# B&R Automation Studio project SDCAxis (part 2)

#### gmcipiec.cnc
```
Root (LangModule=ailgcode, Version=1.0)
  AxesSpec
  PrimTypes (PatternSuffix=:[^\d\w$#])
    BOOL (BRType=BOOL)
    STRING (BRType=STRING)
    WSTRING (BRType=WSTRING)
    TIME (BRType=TIME)
    SINT (BRType=SINT)
    INT (BRType=INT)
    DINT (BRType=DINT)
    USINT (BRType=USINT)
    UINT (BRType=UINT)
    UDINT (BRType=UDINT)
    REAL (BRType=REAL)
    LREAL (BRType=LREAL)
    DATE (BRType=DATE)
    DATE_AND_TIME (BRType=DATE_AND_TIME)
    DT (BRType=DT)
    TIME_OF_DAY (BRType=TIME_OF_DAY)
    TOD (BRType=TIME_OF_DAY)
    BYTE (BRType=BYTE)
    WORD (BRType=WORD)
    DWORD (BRType=DWORD)
  BuiltInProcs:
    SetCyclicId = #job->group_id = $[1]; (MinArgs=1, MaxArgs=1, Eval=Early)
    WaitForCyclic = if ( Defined(:$[1]:) ) 
        WaitForCyclicGroups(:${*}:);  
      else
        WaitForCyclicJob(:#last_job_id:);
      endif (MinArgs=0, MaxArgs=*)
    REPORT (MinArgs=2, MaxArgs=2)
      Arg (ref=id, DataType=INT)
      Arg (ref=msg, DataType=STRING)
    WARN (MinArgs=2, MaxArgs=2)
      Arg (ref=id, DataType=INT)
      Arg (ref=msg, DataType=STRING)
    HALT (MinArgs=2, MaxArgs=2)
      Arg (ref=id, DataType=INT)
      Arg (ref=msg, DataType=STRING)
    ERROR (MinArgs=2, MaxArgs=2)
      Arg (ref=id, DataType=INT)
      Arg (ref=msg, DataType=STRING)
    LOADBG (MinArgs=1, MaxArgs=1)
      Arg (ref=filename, DataType=STRING)
    LOAD (MinArgs=1, MaxArgs=1)
      Arg (ref=filename, DataType=STRING)
    UNLOAD (MinArgs=1, MaxArgs=1)
      Arg (ref=filename, DataType=STRING)
    EXEC (MinArgs=1, MaxArgs=5)
      Arg (ref=filename, DataType=STRING)
      Arg (ref=arguments, DataType=ANY_DATA)
      Arg (ref=langId, DataType=INT)
      Arg (ref=block, DataType=INT, MinCount=0, MaxCount=1, DenyArgs=5, WriteOpts=:)
      Arg (ref=line, DataType=INT, MinCount=0, MaxCount=1, DenyArgs=4, WriteOpts=:)
    EXEC_RPC (MinArgs=2, MaxArgs=4)
      Arg (ref=filename, DataType=STRING)
      Arg (ref=arguments, DataType=ANY_DATA)
      Arg (ref=langId, DataType=INT)
      Arg (ref=rpc, DataType=ANY_DATA, MinCount=1, MaxCount=1)
    EVAL (MinArgs=1, MaxArgs=2)
      Arg (ref=expression, DataType=STRING)
      Arg (ref=langId, DataType=INT)
    PUSH_PACKET = PushPacket(::);
    PUSH_PACKET_CMD (MinArgs=1, MaxArgs=2)
      Arg (ref=cmd, DataType=INT)
      Arg (ref=data, DataType=ANY_DATA)
    DISPATCH_AND_WAIT (MinArgs=1, MaxArgs=1)
      Arg (ref=cmd, DataType=INT)
    START_PACKET_LIST = #inhibit_mp_list_dispatch = 1;
    END_PACKET_LIST = #inhibit_mp_list_dispatch = 0;
    LOG_INFO (MinArgs=1, MaxArgs=1)
      Arg (ref=msg, DataType=STRING)
    SET_BLOCK_NUMBER = SetCurBlockNr(:$[1]:); (MinArgs=1, MaxArgs=1)
    SBLOF_PATH = #next_motion.Command = MPCMD_SBL_PATH_INHIBIT;
      PushPacket(::);
    SBLON_PATH = #next_motion.Command = MPCMD_SBL_PATH_RELEASE;
      PushPacket(::);
  BuiltInFns:
    ABS = Abs(:$[1]:) (ReturnType=ANY_NUM, ArgType1=ANY_NUM, Inline=Yes)
    SIN = RSin(:$[1]:) (ReturnType=ANY_REAL, ArgType1=ANY_REAL, Inline=Yes)
    COS = RCos(:$[1]:) (ReturnType=ANY_REAL, ArgType1=ANY_REAL, Inline=Yes)
    TAN = RTan(:$[1]:) (ReturnType=ANY_REAL, ArgType1=ANY_REAL, Inline=Yes)
    ASIN = RASin(:$[1]:) (ReturnType=ANY_REAL, ArgType1=ANY_REAL, Inline=Yes)
    ACOS = RACos(:$[1]:) (ReturnType=ANY_REAL, ArgType1=ANY_REAL, Inline=Yes)
    ATAN = RATan(:$[1]:) (ReturnType=ANY_REAL, ArgType1=ANY_REAL, Inline=Yes)
    SQRT = Sqrt(:$[1]:) (ReturnType=ANY_REAL, ArgType1=ANY_REAL, Inline=Yes)
    LN = Ln(:$[1]:) (ReturnType=ANY_REAL, ArgType1=ANY_REAL, Inline=Yes)
    EXP = Exp(:$[1]:) (ReturnType=ANY_REAL, ArgType1=ANY_REAL, Inline=Yes)
    LOG = Log(:$[1]:) (ReturnType=ANY_REAL, ArgType1=ANY_REAL, Inline=Yes)
    EXPT = Pow(:$[1],$[2]:) (ReturnType=ANY_REAL, ArgType1=ANY_REAL, ArgType2=ANY_NUM, Inline=Yes)
    TRUNC = ToInt(:Fix(:$[1]:):) (ReturnType=IEC_INT, ArgType1=ANY_REAL, Inline=Yes)
    ADR = Adr(:\$[1]:) (ReturnType=IEC_UDINT, ArgType1=ANY_DATA, Inline=Yes)
    REF = \$[1] (ReturnType=ANY_DATA, ArgType1=ANY_DATA, Inline=Yes)
    SIZEOF = Sizeof(:\$[1]:) (ReturnType=IEC_UINT, NumArgs=1, Inline=Yes)
    LIMIT (ReturnType=ANY_NUM, Inline=No)
      Arg (ref=MIN, DataType=ANY_NUM)
      Arg (ref=IN, DataType=ANY_NUM)
      Arg (ref=MAX, DataType=ANY_NUM)
    MIN (ReturnType=ANY_NUM, Inline=No)
      Arg (ref=IN1, DataType=ANY_NUM)
      Arg (ref=IN2, DataType=ANY_NUM)
    MAX (ReturnType=ANY_NUM, Inline=No)
      Arg (ref=IN1, DataType=ANY_NUM)
      Arg (ref=IN2, DataType=ANY_NUM)
    ROL = BitRotL(:$[1],$[2]:) (ReturnType=ANY_NUM, ArgType1=ANY_NUM, ArgType2=IEC_SINT)
    ROR = BitRotR(:$[1],$[2]:) (ReturnType=ANY_NUM, ArgType1=ANY_NUM, ArgType2=IEC_SINT)
    SHR = BitShR(:$[1],$[2]:) (ReturnType=ANY_NUM, ArgType1=ANY_NUM, ArgType2=IEC_SINT)
    SHL = BitShL(:$[1],$[2]:) (ReturnType=ANY_NUM, ArgType1=ANY_NUM, ArgType2=IEC_SINT)
    BIT_TST = AsBitTst(:$[1],$[2]:) (ReturnType=ANY_NUM, ArgType1=ANY_NUM, ArgType2=IEC_SINT)
    BIT_SET = AsBitSet(:$[1],$[2]:) (ReturnType=ANY_NUM, ArgType1=ANY_NUM, ArgType2=IEC_SINT)
    BIT_CLR = AsBitClr(:$[1],$[2]:) (ReturnType=ANY_NUM, ArgType1=ANY_NUM, ArgType2=IEC_SINT)
    TO_BOOL = ToBool(:$[1]:) (ReturnType=IEC_BOOL, ArgType1=ANY_DATA, Inline=Yes)
    TO_USINT = ToUInt(:$[1],1:) (ReturnType=IEC_USINT, ArgType1=ANY_DATA, Inline=Yes)
    TO_BYTE = ToUInt(:$[1],1:) (ReturnType=IEC_BYTE, ArgType1=ANY_DATA, Inline=Yes)
    TO_SINT = ToInt(:$[1],1:) (ReturnType=IEC_SINT, ArgType1=ANY_DATA, Inline=Yes)
    TO_UINT = ToUInt(:$[1],2:) (ReturnType=IEC_UINT, ArgType1=ANY_DATA, Inline=Yes)
    TO_WORD = ToUInt(:$[1],2:) (ReturnType=IEC_WORD, ArgType1=ANY_DATA, Inline=Yes)
    TO_INT = ToInt(:$[1],2:) (ReturnType=IEC_INT, ArgType1=ANY_DATA, Inline=Yes)
    TO_UDINT = ToUInt(:$[1]:) (ReturnType=IEC_UDINT, ArgType1=ANY_DATA, Inline=Yes)
    TO_DWORD = ToUInt(:$[1]:) (ReturnType=IEC_DWORD, ArgType1=ANY_DATA, Inline=Yes)
    TO_DINT = ToInt(:$[1]:) (ReturnType=IEC_DINT, ArgType1=ANY_DATA, Inline=Yes)
    TO_TIME = ToTime(:$[1]:) (ReturnType=IEC_TIME, ArgType1=ANY_DATA, Inline=Yes)
    TO_DT = ToDT(:$[1]:) (ReturnType=IEC_DT, ArgType1=ANY_DATA, Inline=Yes)
    TO_DATE_AND_TIME = ToDT(:$[1]:) (ReturnType=IEC_DT, ArgType1=ANY_DATA, Inline=Yes)
    TO_TOD = ToTOD(:$[1]:) (ReturnType=IEC_TOD, ArgType1=ANY_DATA, Inline=Yes)
    TO_TIME_OF_DAY = ToTOD(:$[1]:) (ReturnType=IEC_TOD, ArgType1=ANY_DATA, Inline=Yes)
    TO_DATE = ToDate(:$[1]:) (ReturnType=IEC_DATE, ArgType1=ANY_DATA, Inline=Yes)
    TO_REAL = ToFloat(:$[1]:) (ReturnType=IEC_REAL, ArgType1=ANY_DATA, Inline=Yes)
    TO_LREAL = ToLReal(:$[1]:) (ReturnType=IEC_LREAL, ArgType1=ANY_DATA, Inline=Yes)
    TO_STRING = ToString(:$[1]:) (ReturnType=IEC_STRING, ArgType1=ANY_DATA, Inline=Yes)
    TO_WSTRING = ToWString(:$[1]:) (ReturnType=IEC_WSTRING, ArgType1=ANY_DATA, Inline=Yes)
    USINT_TO_BOOL = ToBool(:$[1]:) (ReturnType=IEC_BOOL, ArgType1=IEC_USINT, Inline=Yes)
    SINT_TO_BOOL = ToBool(:$[1]:) (ReturnType=IEC_BOOL, ArgType1=IEC_SINT, Inline=Yes)
    UINT_TO_BOOL = ToBool(:$[1]:) (ReturnType=IEC_BOOL, ArgType1=IEC_UINT, Inline=Yes)
    INT_TO_BOOL = ToBool(:$[1]:) (ReturnType=IEC_BOOL, ArgType1=IEC_INT, Inline=Yes)
    UDINT_TO_BOOL = ToBool(:$[1]:) (ReturnType=IEC_BOOL, ArgType1=IEC_UDINT, Inline=Yes)
    DINT_TO_BOOL = ToBool(:$[1]:) (ReturnType=IEC_BOOL, ArgType1=IEC_DINT, Inline=Yes)
    REAL_TO_BOOL = ToBool(:$[1]:) (ReturnType=IEC_BOOL, ArgType1=IEC_REAL, Inline=Yes)
    LREAL_TO_BOOL = ToBool(:$[1]:) (ReturnType=IEC_BOOL, ArgType1=IEC_LREAL, Inline=Yes)
    TIME_TO_BOOL = ToBool(:$[1]:) (ReturnType=IEC_BOOL, ArgType1=IEC_TIME, Inline=Yes)
    DT_TO_BOOL = ToBool(:$[1]:) (ReturnType=IEC_BOOL, ArgType1=IEC_DT, Inline=Yes)
    TOD_TO_BOOL = ToBool(:$[1]:) (ReturnType=IEC_BOOL, ArgType1=IEC_TOD, Inline=Yes)
    BYTE_TO_BOOL = ToBool(:$[1]:) (ReturnType=IEC_BOOL, ArgType1=IEC_BYTE, Inline=Yes)
    WORD_TO_BOOL = ToBool(:$[1]:) (ReturnType=IEC_BOOL, ArgType1=IEC_WORD, Inline=Yes)
    DWORD_TO_BOOL = ToBool(:$[1]:) (ReturnType=IEC_BOOL, ArgType1=IEC_DWORD, Inline=Yes)
    BOOL_TO_USINT = ToUInt(:$[1],1:) (ReturnType=IEC_USINT, ArgType1=IEC_BOOL, Inline=Yes)
    SINT_TO_USINT = ToUInt(:$[1],1:) (ReturnType=IEC_USINT, ArgType1=IEC_SINT, Inline=Yes)
    UINT_TO_USINT = ToUInt(:$[1],1:) (ReturnType=IEC_USINT, ArgType1=IEC_UINT, Inline=Yes)
    INT_TO_USINT = ToUInt(:$[1],1:) (ReturnType=IEC_USINT, ArgType1=IEC_INT, Inline=Yes)
    UDINT_TO_USINT = ToUInt(:$[1],1:) (ReturnType=IEC_USINT, ArgType1=IEC_UDINT, Inline=Yes)
    DINT_TO_USINT = ToUInt(:$[1],1:) (ReturnType=IEC_USINT, ArgType1=IEC_DINT, Inline=Yes)
    REAL_TO_USINT = ToUInt(:$[1],1:) (ReturnType=IEC_USINT, ArgType1=IEC_REAL, Inline=Yes)
    LREAL_TO_USINT = ToUInt(:$[1],1:) (ReturnType=IEC_USINT, ArgType1=IEC_LREAL, Inline=Yes)
    BOOL_TO_SINT = ToInt(:$[1],1:) (ReturnType=IEC_SINT, ArgType1=IEC_BOOL, Inline=Yes)
    USINT_TO_SINT = ToInt(:$[1],1:) (ReturnType=IEC_SINT, ArgType1=IEC_USINT, Inline=Yes)
    UINT_TO_SINT = ToInt(:$[1],1:) (ReturnType=IEC_SINT, ArgType1=IEC_UINT, Inline=Yes)
    INT_TO_SINT = ToInt(:$[1],1:) (ReturnType=IEC_SINT, ArgType1=IEC_INT, Inline=Yes)
    UDINT_TO_SINT = ToInt(:$[1],1:) (ReturnType=IEC_SINT, ArgType1=IEC_UDINT, Inline=Yes)
    DINT_TO_SINT = ToInt(:$[1],1:) (ReturnType=IEC_SINT, ArgType1=IEC_DINT, Inline=Yes)
    REAL_TO_SINT = ToInt(:$[1],1:) (ReturnType=IEC_SINT, ArgType1=IEC_REAL, Inline=Yes)
    LREAL_TO_SINT = ToInt(:$[1],1:) (ReturnType=IEC_SINT, ArgType1=IEC_LREAL, Inline=Yes)
    BOOL_TO_UINT = ToUInt(:$[1],2:) (ReturnType=IEC_UINT, ArgType1=IEC_BOOL, Inline=Yes)
    SINT_TO_UINT = ToUInt(:$[1],2:) (ReturnType=IEC_UINT, ArgType1=IEC_SINT, Inline=Yes)
    USINT_TO_UINT = ToUInt(:$[1],2:) (ReturnType=IEC_UINT, ArgType1=IEC_USINT, Inline=Yes)
    INT_TO_UINT = ToUInt(:$[1],2:) (ReturnType=IEC_UINT, ArgType1=IEC_INT, Inline=Yes)
    UDINT_TO_UINT = ToUInt(:$[1],2:) (ReturnType=IEC_UINT, ArgType1=IEC_UDINT, Inline=Yes)
    DINT_TO_UINT = ToUInt(:$[1],2:) (ReturnType=IEC_UINT, ArgType1=IEC_DINT, Inline=Yes)
    REAL_TO_UINT = ToUInt(:$[1],2:) (ReturnType=IEC_UINT, ArgType1=IEC_REAL, Inline=Yes)
    LREAL_TO_UINT = ToUInt(:$[1],2:) (ReturnType=IEC_UINT, ArgType1=IEC_LREAL, Inline=Yes)
    BOOL_TO_INT = ToInt(:$[1],2:) (ReturnType=IEC_INT, ArgType1=IEC_BOOL, Inline=Yes)
    SINT_TO_INT = ToInt(:$[1],2:) (ReturnType=IEC_INT, ArgType1=IEC_SINT, Inline=Yes)
    USINT_TO_INT = ToInt(:$[1],2:) (ReturnType=IEC_INT, ArgType1=IEC_USINT, Inline=Yes)
    UINT_TO_INT = ToInt(:$[1],2:) (ReturnType=IEC_INT, ArgType1=IEC_UINT, Inline=Yes)
    UDINT_TO_INT = ToInt(:$[1],2:) (ReturnType=IEC_INT, ArgType1=IEC_UDINT, Inline=Yes)
    DINT_TO_INT = ToInt(:$[1],2:) (ReturnType=IEC_INT, ArgType1=IEC_DINT, Inline=Yes)
    REAL_TO_INT = ToInt(:$[1],2:) (ReturnType=IEC_INT, ArgType1=IEC_REAL, Inline=Yes)
    LREAL_TO_INT = ToInt(:$[1],2:) (ReturnType=IEC_INT, ArgType1=IEC_LREAL, Inline=Yes)
    BOOL_TO_UDINT = ToUInt(:$[1]:) (ReturnType=IEC_UDINT, ArgType1=IEC_BOOL, Inline=Yes)
    USINT_TO_UDINT = ToUInt(:$[1]:) (ReturnType=IEC_UDINT, ArgType1=IEC_USINT, Inline=Yes)
    SINT_TO_UDINT = ToUInt(:$[1]:) (ReturnType=IEC_UDINT, ArgType1=IEC_SINT, Inline=Yes)
    UINT_TO_UDINT = ToUInt(:$[1]:) (ReturnType=IEC_UDINT, ArgType1=IEC_UINT, Inline=Yes)
    INT_TO_UDINT = ToUInt(:$[1]:) (ReturnType=IEC_UDINT, ArgType1=IEC_INT, Inline=Yes)
    DINT_TO_UDINT = ToUInt(:$[1]:) (ReturnType=IEC_UDINT, ArgType1=IEC_DINT, Inline=Yes)
    REAL_TO_UDINT = ToUInt(:$[1]:) (ReturnType=IEC_UDINT, ArgType1=IEC_REAL, Inline=Yes)
    LREAL_TO_UDINT = ToUInt(:$[1]:) (ReturnType=IEC_UDINT, ArgType1=IEC_LREAL, Inline=Yes)
    TIME_TO_UDINT = ToUInt(:$[1]:) (ReturnType=IEC_UDINT, ArgType1=IEC_TIME, Inline=Yes)
    DT_TO_UDINT = ToUInt(:$[1]:) (ReturnType=IEC_UDINT, ArgType1=IEC_DT, Inline=Yes)
    BOOL_TO_DINT = ToInt(:$[1]:) (ReturnType=IEC_DINT, ArgType1=IEC_BOOL, Inline=Yes)
    USINT_TO_DINT = ToInt(:$[1]:) (ReturnType=IEC_DINT, ArgType1=IEC_USINT, Inline=Yes)
    SINT_TO_DINT = ToInt(:$[1]:) (ReturnType=IEC_DINT, ArgType1=IEC_SINT, Inline=Yes)
    UINT_TO_DINT = ToInt(:$[1]:) (ReturnType=IEC_DINT, ArgType1=IEC_UINT, Inline=Yes)
    INT_TO_DINT = ToInt(:$[1]:) (ReturnType=IEC_DINT, ArgType1=IEC_INT, Inline=Yes)
    UDINT_TO_DINT = ToInt(:$[1]:) (ReturnType=IEC_DINT, ArgType1=IEC_UDINT, Inline=Yes)
    REAL_TO_DINT = ToInt(:$[1]:) (ReturnType=IEC_DINT, ArgType1=IEC_REAL, Inline=Yes)
    LREAL_TO_DINT = ToInt(:$[1]:) (ReturnType=IEC_DINT, ArgType1=IEC_LREAL, Inline=Yes)
    TIME_TO_DINT = ToInt(:$[1]:) (ReturnType=IEC_DINT, ArgType1=IEC_TIME, Inline=Yes)
    DT_TO_DINT = ToInt(:$[1]:) (ReturnType=IEC_DINT, ArgType1=IEC_DT, Inline=Yes)
    BOOL_TO_TIME = ToTime(:$[1]:) (ReturnType=IEC_TIME, ArgType1=IEC_BOOL, Inline=Yes)
    DINT_TO_TIME = ToTime(:$[1]:) (ReturnType=IEC_TIME, ArgType1=IEC_DINT, Inline=Yes)
    UDINT_TO_TIME = ToTime(:$[1]:) (ReturnType=IEC_TIME, ArgType1=IEC_UDINT, Inline=Yes)
    BOOL_TO_DT = ToDT(:$[1]:) (ReturnType=IEC_DT, ArgType1=IEC_BOOL, Inline=Yes)
    DINT_TO_DT = ToDT(:$[1]:) (ReturnType=IEC_DT, ArgType1=IEC_DINT, Inline=Yes)
    UDINT_TO_DT = ToDT(:$[1]:) (ReturnType=IEC_DT, ArgType1=IEC_UDINT, Inline=Yes)
    BOOL_TO_REAL = ToFloat(:$[1]:) (ReturnType=IEC_REAL, ArgType1=IEC_BOOL, Inline=Yes)
    USINT_TO_REAL = ToFloat(:$[1]:) (ReturnType=IEC_REAL, ArgType1=IEC_USINT, Inline=Yes)
    SINT_TO_REAL = ToFloat(:$[1]:) (ReturnType=IEC_REAL, ArgType1=IEC_SINT, Inline=Yes)
    UINT_TO_REAL = ToFloat(:$[1]:) (ReturnType=IEC_REAL, ArgType1=IEC_UINT, Inline=Yes)
    INT_TO_REAL = ToFloat(:$[1]:) (ReturnType=IEC_REAL, ArgType1=IEC_INT, Inline=Yes)
    UDINT_TO_REAL = ToFloat(:$[1]:) (ReturnType=IEC_REAL, ArgType1=IEC_UDINT, Inline=Yes)
    DINT_TO_REAL = ToFloat(:$[1]:) (ReturnType=IEC_REAL, ArgType1=IEC_DINT, Inline=Yes)
    LREAL_TO_REAL = ToFloat(:$[1]:) (ReturnType=IEC_REAL, ArgType1=IEC_LREAL, Inline=Yes)
    TIME_TO_REAL = ToFloat(:$[1]:) (ReturnType=IEC_REAL, ArgType1=IEC_TIME, Inline=Yes)
    BOOL_TO_LREAL = ToLReal(:$[1]:) (ReturnType=IEC_LREAL, ArgType1=IEC_BOOL, Inline=Yes)
    USINT_TO_LREAL = ToLReal(:$[1]:) (ReturnType=IEC_LREAL, ArgType1=IEC_USINT, Inline=Yes)
    SINT_TO_LREAL = ToLReal(:$[1]:) (ReturnType=IEC_LREAL, ArgType1=IEC_SINT, Inline=Yes)
    UINT_TO_LREAL = ToLReal(:$[1]:) (ReturnType=IEC_LREAL, ArgType1=IEC_UINT, Inline=Yes)
    INT_TO_LREAL = ToLReal(:$[1]:) (ReturnType=IEC_LREAL, ArgType1=IEC_INT, Inline=Yes)
    UDINT_TO_LREAL = ToLReal(:$[1]:) (ReturnType=IEC_LREAL, ArgType1=IEC_UDINT, Inline=Yes)
    DINT_TO_LREAL = ToLReal(:$[1]:) (ReturnType=IEC_LREAL, ArgType1=IEC_DINT, Inline=Yes)
    REAL_TO_LREAL = ToLReal(:$[1]:) (ReturnType=IEC_LREAL, ArgType1=IEC_REAL, Inline=Yes)
    TIME_TO_LREAL = ToLReal(:$[1]:) (ReturnType=IEC_LREAL, ArgType1=IEC_TIME, Inline=Yes)
    BOOL_TO_STRING = ToString(:ToBool(:$[1]:):) (ReturnType=IEC_STRING, ArgType1=IEC_BOOL, Inline=Yes)
    USINT_TO_STRING = ToString(:ToUInt(:$[1],1:):) (ReturnType=IEC_STRING, ArgType1=IEC_USINT, Inline=Yes)
    SINT_TO_STRING = ToString(:ToInt(:$[1],1:):) (ReturnType=IEC_STRING, ArgType1=IEC_SINT, Inline=Yes)
    UINT_TO_STRING = ToString(:ToUInt(:$[1],2:):) (ReturnType=IEC_STRING, ArgType1=IEC_UINT, Inline=Yes)
    INT_TO_STRING = ToString(:ToInt(:$[1],2:):) (ReturnType=IEC_STRING, ArgType1=IEC_INT, Inline=Yes)
    UDINT_TO_STRING = ToString(:ToUInt(:$[1]:):) (ReturnType=IEC_STRING, ArgType1=IEC_UDINT, Inline=Yes)
    DINT_TO_STRING = ToString(:ToInt(:$[1]:):) (ReturnType=IEC_STRING, ArgType1=IEC_DINT, Inline=Yes)
    REAL_TO_STRING = ToString(:ToFloat(:$[1]:):) (ReturnType=IEC_STRING, ArgType1=IEC_REAL, Inline=Yes)
    LREAL_TO_STRING = ToString(:ToLReal(:$[1]:):) (ReturnType=IEC_STRING, ArgType1=IEC_LREAL, Inline=Yes)
    STRING_TO_BOOL = ToBool(:StrToInt(:$[1]:):) (ReturnType=IEC_BOOL, ArgType1=IEC_STRING, Inline=Yes)
    STRING_TO_USINT = ToUInt(:StrToInt(:$[1]:),1:) (ReturnType=IEC_USINT, ArgType1=IEC_STRING, Inline=Yes)
    STRING_TO_SINT = ToInt(:StrToInt(:$[1]:),1:) (ReturnType=IEC_SINT, ArgType1=IEC_STRING, Inline=Yes)
    STRING_TO_UINT = ToUInt(:StrToInt(:$[1]:),2:) (ReturnType=IEC_UINT, ArgType1=IEC_STRING, Inline=Yes)
    STRING_TO_INT = ToInt(:StrToInt(:$[1]:),2:) (ReturnType=IEC_INT, ArgType1=IEC_STRING, Inline=Yes)
    STRING_TO_UDINT = ToUInt(:StrToInt(:$[1]:):) (ReturnType=IEC_UDINT, ArgType1=IEC_STRING, Inline=Yes)
    STRING_TO_DINT = ToInt(:StrToInt(:$[1]:):) (ReturnType=IEC_DINT, ArgType1=IEC_STRING, Inline=Yes)
    STRING_TO_REAL = ToFloat(:ToLReal(:$[1]:):) (ReturnType=IEC_REAL, ArgType1=IEC_STRING, Inline=Yes)
    STRING_TO_LREAL = ToLReal(:$[1]:) (ReturnType=IEC_LREAL, ArgType1=IEC_STRING, Inline=Yes)
    LEN = __LEN(:$[1]:) (ReturnType=IEC_INT, ArgType1=IEC_STRING, Inline=Yes)
    LEFT = __LEFT(:$[1], $[2]:) (ReturnType=IEC_STRING, ArgType1=IEC_STRING, ArgType2=IEC_INT, Inline=Yes)
    RIGHT = __RIGHT(:$[1], $[2]:) (ReturnType=IEC_STRING, ArgType1=IEC_STRING, ArgType2=IEC_INT, Inline=Yes)
    MID = __MID(:$[1], $[2], $[3]:) (ReturnType=IEC_STRING, ArgType1=IEC_STRING, ArgType2=IEC_INT, ArgType3=IEC_INT, Inline=Yes)
    CONCAT = __CONCAT(:$[1], $[2]:) (ReturnType=IEC_STRING, ArgType1=IEC_STRING, ArgType2=IEC_STRING, Inline=Yes)
    INSERT = __INSERT(:$[1], $[2], $[3]:) (ReturnType=IEC_STRING, ArgType1=IEC_STRING, ArgType2=IEC_STRING, ArgType3=IEC_INT, Inline=Yes)
    DELETE = __DELETE(:$[1], $[2], $[3]:) (ReturnType=IEC_STRING, ArgType1=IEC_STRING, ArgType2=IEC_INT, ArgType3=IEC_INT, Inline=Yes)
    REPLACE = __REPLACE(:$[1], $[2], $[3], $[4]:) (ReturnType=IEC_STRING, ArgType1=IEC_STRING, ArgType2=IEC_STRING, ArgType3=IEC_INT, ArgType4=IEC_INT, Inline=Yes)
    FIND = __FIND(:$[1], $[2]:) (ReturnType=IEC_INT, ArgType1=IEC_STRING, ArgType2=IEC_STRING, Inline=Yes)
    IP_INST_NUM = IpInstNum(::) (ReturnType=IEC_INT, NumArgs=0)
    IP_OWNER_ID = IpOwnerId(::) (ReturnType=IEC_INT, NumArgs=0)
    PACKET_DATA_ADR = GetIpInt(:6:) (ReturnType=IEC_UDINT, NumArgs=0, Inline=Yes)
    PACKET_COMMAND_ADR = GetIpInt(:7:) (ReturnType=IEC_UDINT, NumArgs=0, Inline=Yes)
  Parameters:
    QUOTED (QuotedName=$R, ValueType=FLOAT, ReturnType=IEC_LREAL)
      ARG (ref=EXPR, DataType=INT, MinValue=0, MaxValue=999)
    QUOTED (QuotedName=$P, ValueType=FLOAT, ReturnType=IEC_LREAL)
      ARG (ref=EXPR, DataType=INT, MinValue=0, MaxValue=999)
    QUOTED (QuotedName=$EXB, ValueType=INT, ReturnType=IEC_SINT)
      ARG (ref=EXPR, DataType=INT, MinValue=0, MaxValue=99)
    QUOTED (QuotedName=$EXW, ValueType=INT, ReturnType=IEC_INT)
      ARG (ref=EXPR, DataType=INT, MinValue=0, MaxValue=99)
    QUOTED (QuotedName=$EXL, ValueType=INT, ReturnType=IEC_DINT)
      ARG (ref=EXPR, DataType=INT, MinValue=0, MaxValue=99)
    QUOTED (QuotedName=$EXF, ValueType=FLOAT, ReturnType=IEC_REAL)
      ARG (ref=EXPR, DataType=INT, MinValue=0, MaxValue=3999)
    QUOTED (QuotedName=$MW, Synchronous=Yes, ValueType=INT, ReturnType=IEC_INT)
      ARG (ref=EXPR, DataType=INT, MinValue=0, MaxValue=99)
    QUOTED (QuotedName=$ML, Synchronous=Yes, ValueType=INT, ReturnType=IEC_DINT)
      ARG (ref=EXPR, DataType=INT, MinValue=0, MaxValue=99)
    QUOTED (QuotedName=$MF, Synchronous=Yes, ValueType=FLOAT, ReturnType=IEC_REAL)
      ARG (ref=EXPR, DataType=INT, MinValue=0, MaxValue=99)
  ParserData (NestedComments=No, DefaultCaseSensitive=Yes, CommentsSpanLines=Yes, ReadWholeFileBeforeParsing=Yes, ExpectMainProgStmts=No, UseFubTemplates=No, LexerType=IEC, RuntimePreventOverflow=No, RoundRealToInt=No, AllowArrayRefWithoutIndex=Yes, DeclareEnumLiteralsAsConstants=No, AllowVariableAutoDereference=Yes, AllowStructMemberAutoDereference=No, AllowPassByRefFnArgAutoReference=No, AllowNamedFnArgs=Yes, AllowUnnamedFnArgs=Yes, AllowFnArgMixedNaming=Yes, AllowFnArgsOutOfSequence=No, AllowBuiltinFnArgsOutOfSequence=Yes, AllowFnArgsOmmitted=Yes, AllowIgnoredFnReturn=Yes, AllowIgnoredExtraSubArgs=No, AllowFnStringInputArgsShort=No, RefuseBuiltinFnUnknownArgName=Yes, AllowBuiltinFnArgCaseSensitive=Yes)
    TKG_OPEN_COMMENT = (*
    TKG_CLOSE_COMMENT = *)
    TKG_IEC_LINE_COMMENT = //
    TKG_TRUE = TRUE:[^\w\d] (IsPattern=Yes)
    TKG_FALSE = FALSE:[^\w\d] (IsPattern=Yes)
    TKG_PRIM_TYPE (IsPattern=Yes)
    TKG_OPEN_BRACKET = (
    TKG_CLOSE_BRACKET = )
    TKG_OPEN_INDEXBRACKET = [
    TKG_CLOSE_INDEXBRACKET = ]
    TKG_COMMA = ,
    TKG_SUBRANGE = ..
    TKG_IEC_BINARY_INTEGER = 2#_[01][01_]+|2#[01][01_]+|2#_[01]|2#[01] (IsPattern=Yes)
    TKG_IEC_OCTAL_INTEGER = 8#_[0-7][0-7_]+|8#[0-7][0-7_]+|8#_[0-7]|8#[0-7] (IsPattern=Yes)
    TKG_IEC_HEX_INTEGER = 16#_[\da-fA-F][\da-fA-F]+|16#[\da-fA-F][\da-fA-F_]+|16#_[\da-fA-F]|16#[\da-fA-F] (IsPattern=Yes)
    TKG_REAL = \d[\d_]*\.[\d_]+[Ee][\+\-]\d[\d_]*|\d[\d_]*\.[\d_]+[Ee]\d[\d_]*|\d[\d_]*\.[\d_]+ (IsPattern=Yes)
    TKG_REAL_EXP = \d[\d_]*[Ee]\d[\d_]*|\d[\d_]*[Ee][\+\-]\d[\d_]* (IsPattern=Yes)
    TKG_INTEGER = \d|\d[\d_]+ (IsPattern=Yes)
    TKG_DOT = .
    TKG_PATHSYNCH_REC_IEC = DO_PATH_SYNCH:[^\w\d] (IsPattern=Yes, EndRuleToken=Yes)
    TKG_PATHSYNCH_END = END_PATH_SYNCH:[^\w\d] (IsPattern=Yes, EndRuleToken=Yes)
    TKG_PATHSYNCH_IPEVAL = IP_EVAL:[^\w\d] (IsPattern=Yes)
    TKG_CYCLIC_PATHSYNCH_BLOCKING_IEC = CYCLIC_PS_BL:[^\w\d] (IsPattern=Yes, EndRuleToken=Yes)
    TKG_CYCLIC_PATHSYNCH_IEC = CYCLIC_PS:[^\w\d] (IsPattern=Yes, EndRuleToken=Yes)
    TKG_CYCLIC_BLOCKING_IEC = CYCLIC_BL:[^\w\d] (IsPattern=Yes, EndRuleToken=Yes)
    TKG_CYCLIC_IEC = CYCLIC:[^\w\d] (IsPattern=Yes, EndRuleToken=Yes)
    TKG_CYCLIC_END_IEC = END_CYCLIC:[^\w\d] (IsPattern=Yes, EndRuleToken=Yes)
    TKG_REFERENCE = REFERENCE:[^\w\d] (FollowedBy=TKG_IEC_TO, IsPattern=Yes)
    TKG_IEC_TO = TO:[^\w\d] (IsPattern=Yes)
    TKG_IEC_DO = DO:[^\w\d] (IsPattern=Yes, EndRuleToken=Yes)
    TKG_FOR_NOFINALDEC = FOR:[^\w\d] (FileXLInvalid=Yes, IsPattern=Yes)
    TKG_FORSTEP = BY:[^\w\d] (FileXLInvalid=Yes, IsPattern=Yes)
    TKG_ENDFOR = END_FOR:[^\w\d] (FileXLInvalid=Yes, IsPattern=Yes, EndRuleToken=Yes)
    TKG_IF = IF:[^\w\d] (IsPattern=Yes)
    TKG_THEN = THEN:[^\w\d] (IsPattern=Yes, EndRuleToken=Yes)
    TKG_BLOCK_ELSEIF = ELSIF:[^\w\d] (IsPattern=Yes)
    TKG_ELSE_AND_DEFAULT = ELSE:[^\w\d] (IsPattern=Yes, EndRuleToken=Yes)
    TKG_BLOCK_ENDIF = END_IF:[^\w\d] (IsPattern=Yes, EndRuleToken=Yes)
    TKG_SWITCH = CASE:[^\w\d] (IsPattern=Yes, FileXLInvalid=Yes)
    TKG_ENDSWITCH_NOBREAK = END_CASE:[^\w\d] (FileXLInvalid=Yes, IsPattern=Yes, EndRuleToken=Yes)
    TKG_WHILE = WHILE:[^\w\d] (FileXLInvalid=Yes, IsPattern=Yes)
    TKG_ENDWHILE = END_WHILE:[^\w\d] (FileXLInvalid=Yes, IsPattern=Yes, EndRuleToken=Yes)
    TKG_DO = REPEAT:[^\w\d] (FileXLInvalid=Yes, IsPattern=Yes, EndRuleToken=Yes)
    TKG_ENDDO_UNTIL = UNTIL:[^\w\d] (FileXLInvalid=Yes, IsPattern=Yes)
    TKG_ENDDO_POSTCOND = END_REPEAT:[^\w\d] (FileXLInvalid=Yes, IsPattern=Yes, EndRuleToken=Yes)
    TKG_BREAK = EXIT:[^\w\d] (FileXLInvalid=Yes, IsPattern=Yes)
    TKG_RETURN = RETURN:[^\w\d] (FileXLInvalid=Yes, IsPattern=Yes)
    TKG_IEC_SEL_FN = SEL:[^\w\d] (FileXLInvalid=Yes, IsPattern=Yes)
    TKG_IEC_MUX_FN = MUX:[^\w\d] (FileXLInvalid=Yes, IsPattern=Yes)
    TKG_TIME_LITERAL = time#\-[dDhHmMsS_\.\d]+|time#[dDhHmMsS_\.\d]+|t#\-[dDhHmMsS_\.\d]+|t#[dDhHmMsS_\.\d]+ (CaseSensitive=no, IsPattern=yes)
    TKG_DATE_AND_TIME_LITERAL = DT#[12]\d\d\d\-[\d\:\-]*|DATE_AND_TIME#[12]\d\d\d\-[\d\:\-]* (CaseSensitive=no, IsPattern=yes)
    TKG_DATE_LITERAL = D#[12]\d\d\d\-[\d\-]*|DATE#[12]\d\d\d\-[\d\-]* (CaseSensitive=no, IsPattern=yes)
    TKG_TIME_OF_DAY_LITERAL = TOD#\d[\d\:\.]*|TIME_OF_DAY#\d[\d\:\.]* (CaseSensitive=no, IsPattern=yes)
    TKG_ASSIGN_EQ = :=
    TKG_OPEN_IP_EXTENSION = {
    TKG_CLOSE_IP_EXTENSION = }
    TKG_IEC_OPEN_TYPE = TYPE:[^\w\d] (IsPattern=Yes)
    TKG_IEC_CLOSE_TYPE = END_TYPE:[^\w\d] (IsPattern=Yes, EndRuleToken=Yes)
    TKG_VAR = VAR:[^\w\d] (IsPattern=Yes)
    TKG_VAR_GLOBAL = VAR_GLOBAL:[^\w\d] (IsPattern=Yes)
    TKG_VAR_INPUT = VAR_INPUT:[^\w\d] (IsPattern=Yes)
    TKG_VAR_OUTPUT = VAR_OUTPUT:[^\w\d] (IsPattern=Yes)
    TKG_VAR_IN_OUT = VAR_IN_OUT:[^\w\d] (IsPattern=Yes)
    TKG_VAR_END = END_VAR:[^\w\d] (IsPattern=Yes, EndRuleToken=Yes)
    TKG_VAR_RETAIN = RETAIN:[^\d\w] (IsPattern=Yes)
    TKG_IP_RETAIN = IP_RETAIN:[^\d\w] (IsPattern=Yes)
    TKG_AT = AT:[^\d\w] (IsPattern=Yes)
    TKG_PLC = PLC:[^\d\w] (IsPattern=Yes)
    TKG_PV_UNDECL = UNRETAIN_VAR:[^\d\w] (IsPattern=Yes)
    TKG_VARSYNCH_IP = IP_SYNCH:[^\d\w] (IsPattern=Yes)
    TKG_VARSYNCH_PATH = PATH_SYNCH:[^\d\w] (IsPattern=Yes)
    TKG_CONSTANT = CONSTANT:[^\d\w] (IsPattern=Yes)
    TKG_VARSCOPE_IP_GLOBAL = IP_GLOBAL:[^\w\d] (IsPattern=Yes)
    TKG_VARSCOPE_SHARED_IP_GLOBAL = SHARED_IP_GLOBAL:[^\w\d] (IsPattern=Yes)
    TKG_VARSCOPE_NC_GLOBAL = NC_GLOBAL:[^\w\d] (IsPattern=Yes)
    TKG_VARSCOPE_PLC_GLOBAL = PLC_GLOBAL:[^\w\d] (IsPattern=Yes)
    TKG_VARSCOPE_IP_LOCAL = LOCAL:[^\w\d] (IsPattern=Yes)
    TKG_IEC_NAMESPACE_SPEC = :: (IsPattern=No)
    TKG_IEC_DATATYPE_SPEC = : (IsPattern=No)
    TKG_IEC_ARRAY = ARRAY:[^\w\d] (IsPattern=Yes)
    TKG_IEC_OF = OF:[^\w\d] (IsPattern=Yes)
    TKG_IEC_DELIM = ; (EndRuleToken=Yes)
    TKG_IEC_OPEN_STRUCT = STRUCT:[^\w\d] (IsPattern=Yes)
    TKG_IEC_CLOSE_STRUCT = END_STRUCT:[^\w\d] (IsPattern=Yes)
    TKG_BITWISE_LP_BINARY_AND = AND:[^\w\d] (IsPattern=Yes)
    TKG_BITWISE_LP_BINARY_OR = OR:[^\w\d] (IsPattern=Yes)
    TKG_BITWISE_LP_BINARY_XOR = XOR:[^\w\d] (IsPattern=Yes)
    TKG_BITWISE_UNARY_COMPLEMENT = NOT:[^\w\d] (IsPattern=Yes)
    TKG_COMP_EXACT_BINARY_GREATER_THAN_OR_EQ = >=
    TKG_COMP_EXACT_BINARY_LESS_THAN_OR_EQ = <=
    TKG_COMP_EXACT_BINARY_EQUAL_TO = =
    TKG_COMP_EXACT_BINARY_NOT_EQUAL_TO = <>
    TKG_COMP_EXACT_BINARY_GREATER_THAN = >
    TKG_COMP_EXACT_BINARY_LESS_THAN = <
    TKG_ARITH_BINARY_PLUS = +
    TKG_ARITH_BINARY_MINUS = -
    TKG_ARITH_BINARY_POWER = **
    TKG_ARITH_BINARY_MULTIPLY = *
    TKG_ARITH_BINARY_DIVIDE = /
    TKG_ARITH_BINARY_MODULO = MOD:[^\w\d] (IsPattern=Yes)
    TKG_PRAGMA = #pragma:[^\w\d] (IsPattern=Yes, FollowedBy=TKG_IDENTIFIER)
    TKG_INCLUDE = #include:[^\w\d] (IsPattern=Yes)
    TKG_PROG_START = PROGRAM:[^\w\d] (IsPattern=Yes, FollowedBy=TKG_PROG_NAME)
    TKG_PROG_NAME = _INIT:[^\w\d]|_CYCLIC:[^\w\d]|_EXIT:[^\w\d]|_MAIN:[^\w\d]|_\d+:[^\w\d] (IsPattern=Yes, EndRuleToken=Yes)
    TKG_PROG_END = END_PROGRAM:[^\w\d] (IsPattern=Yes, EndRuleToken=Yes)
    TKG_SUBPROG_START = FUNCTION:[^\w\d] (IsPattern=Yes)
    TKG_SUBPROG_END = END_FUNCTION:[^\w\d] (IsPattern=Yes, EndRuleToken=Yes)
    TKG_FUB_DECL = FUNCTION_BLOCK:[^\w\d] (IsPattern=Yes)
    TKG_FUB_END = END_FUNCTION_BLOCK:[^\w\d] (IsPattern=Yes, EndRuleToken=Yes)
    TKG_RETURN = RETURN:[^\w\d] (IsPattern=Yes)
    TKG_ACCESS = ACCESS:[^\w\d] (IsPattern=Yes)
    TKG_DEREF_OP = ^
    TKG_ACTION = ACTION:[^\w\d] (IsPattern=Yes)
    TKG_ACTION_END = END_ACTION:[^\w\d] (IsPattern=Yes, EndRuleToken=Yes)
    TKG_IEC_TYPED_VALUE = \w#:[\w\d\+\-]|\w[\w\d]+#:[\w\d\+\-] (IsPattern=Yes)
    TKG_PARAM_PREFIX = $R:[^\w\d]|$P:[^\w\d]|$MW:[^\w\d]|$ML:[^\w\d]|$MF:[^\w\d]|$EXW:[^\w\d]|$EXL:[^\w\d]|$EXF:[^\w\d]|$EXB:[^\w\d] (IsPattern=Yes)
    TKG_IGNORED_IP_EXTENSION = REDUND_CONTEXT|REDUND_UNREPLICABLE|REDUND_OK (IsPattern=Yes)
    TKG_IDENTIFIER = \w|\w[\w\d$]+|$[\w\d$]+ (IsPattern=Yes)
    TKG_INIT_IDENTIFIER = \w|\w[\w\d$]+|$[\w\d$]+ (IsPattern=Yes, Disabled=Yes)
  StringChars (AsciiStringStart=', AsciiStringEnd=', UTF16StringStart=", UTF16StringEnd=")
    EscapeSeq (Search=$N, CaseSensitive=Yes, ReplaceValue=10)
    EscapeSeq (Search=$n, CaseSensitive=Yes, ReplaceValue=10)
    EscapeSeq (Search=$L, CaseSensitive=Yes, ReplaceValue=10)
    EscapeSeq (Search=$l, CaseSensitive=Yes, ReplaceValue=10)
    EscapeSeq (Search=$P, CaseSensitive=Yes, ReplaceValue=12)
    EscapeSeq (Search=$p, CaseSensitive=Yes, ReplaceValue=12)
    EscapeSeq (Search=$R, CaseSensitive=Yes, ReplaceValue=13)
    EscapeSeq (Search=$r, CaseSensitive=Yes, ReplaceValue=13)
    EscapeSeq (Search=$T, CaseSensitive=Yes, ReplaceValue=9)
    EscapeSeq (Search=$t, CaseSensitive=Yes, ReplaceValue=9)
    EscapeSeq (Search=$', CaseSensitive=Yes, ReplaceStr=')
    EscapeSeq (Search=$", CaseSensitive=Yes, ReplaceStr=")
    EscapeSeq (Search=$[\dA-Fa-f]+, IsPattern=Yes, CaseSensitive=Yes, ReplaceEncodingBase=16)
    EscapeSeq (Search=$$, ReplaceStr=$)
    EscapeSeq (Search=$, ReplaceStr=)
```

### Data object Logical/GmcIpConfig/gmciplog (Cnc, version 5.02.1)

#### gmciplog.cnc
```
Root (LangModule=ailgcode, Version=1.0)
  AxesSpec
  PVMacros:
    DR8:
      REF = #next_motion.Data.R8_value
    DI4:
      REF = #next_motion.Data.I4_value
    DU4:
      REF = #next_motion.Data.UI4_value
    DR8_G211:
      SET = %_CNC.TA = ${EXPR};
       if (%_CNC.TA < 0)
         %_CNC.TA = 0;
       endif
        #next_motion.Data.R8_value = ${EXPR};
    Dlp:
      REF = #next_motion.Data.LinMovement.Position
    Dli:
      SET = #next_motion.Data.LinMovement.Idx[0] = ArrayRep(:(:-1:):);
        #next_motion.Data.LinMovement.Idx = ${EXPR};
    Dlm:
      SET = #next_motion.Data.LinMovement.Mode[0] = ArrayRep(:(:-1:):);
        #next_motion.Data.LinMovement.Mode = ${EXPR};
    Dto:
      REF = #next_motion.Data.Trans.Offset
    Dti:
      SET = #next_motion.Data.Trans.AxIdx[0] = ArrayRep(:(:-1:):);
        #next_motion.Data.Trans.AxIdx = ${EXPR};
    Dtm:
      SET = #next_motion.Data.Trans.Mode[0] = ArrayRep(:(:-1:):);
        #next_motion.Data.Trans.Mode = ${EXPR};
    DSPp:
      REF = #next_motion.Data.SplinePoint.Position
    DSPi:
      SET = #next_motion.Data.SplinePoint.AxIdx[0] = ArrayRep(:(:-1:):);
        #next_motion.Data.SplinePoint.AxIdx = ${EXPR};
    DSPm:
      SET = #next_motion.Data.SplinePoint.Mode[0] = ArrayRep(:(:-1:):);
        #next_motion.Data.SplinePoint.Mode = ${EXPR};
    Dcp:
      REF = #next_motion.Data.CircMovement.Parameter
    Dci:
      SET = #next_motion.Data.CircMovement.Idx[0] = ArrayRep(:(:-1:):);
        #next_motion.Data.CircMovement.Idx = ${EXPR};
    Dcm:
      SET = #next_motion.Data.CircMovement.Mode[0] = ArrayRep(:(:-1:):);
        #next_motion.Data.CircMovement.Mode = ${EXPR};
    Dtp:
      REF = #next_motion.Data.ToolAxOrient.Parameter
    Dts:
      REF = #next_motion.Data.ToolAxOrient.Sign
    Daz:
      REF = #next_motion.Data.AbsZeroPtShift.ZpRecIdx
    Das:
      REF = #next_motion.Data.AbsZeroPtShift.SetCS
    Dpt:
      SET = #next_motion.Data.ProgZeroPtShift.Type[0] = ArrayRep(:(:-1:):);
        #next_motion.Data.ProgZeroPtShift.Type = ${EXPR};
    Dpm:
      SET = #next_motion.Data.ProgZeroPtShift.Mode[0] = ArrayRep(:(:-1:):);
        #next_motion.Data.ProgZeroPtShift.Mode = ${EXPR};
    Dpa:
      REF = #next_motion.Data.ProgZeroPtShift.AxShift
    Dovpathdef:
      REF = #next_motion.Data.OptMotPar.path_definition
    Dovpathdefd:
      REF = #next_motion.Data.OptMotPar.path_definition_def
    Dorpar:
      REF = #next_motion.Data.OptMotPar.robot_par
    Dorpard:
      REF = #next_motion.Data.OptMotPar.robot_par_def
    Dolim:
      REF = #next_motion.Data.OptMotPar.limits_idx
    Dolimd:
      REF = #next_motion.Data.OptMotPar.limits_idx_def
    Dolimfac:
      REF = #next_motion.Data.OptMotPar.limits_factor
    Dolimfacd:
      REF = #next_motion.Data.OptMotPar.limits_factor_def
    Dfdx:
      REF = #next_motion.Data.FullTrfTool.Dx
    Dfdy:
      REF = #next_motion.Data.FullTrfTool.Dy
    Dfdz:
      REF = #next_motion.Data.FullTrfTool.Dz
    Dfph:
      REF = #next_motion.Data.FullTrfTool.Phi
    Dft:
      REF = #next_motion.Data.FullTrfTool.Theta
    Dfps:
      REF = #next_motion.Data.FullTrfTool.Psi
    DPLDli:
      REF = #next_motion.Data.PosLatchDistance.LatchIdx
    DPLDts:
      REF = #next_motion.Data.PosLatchDistance.TriggSource
    DPLDe:
      REF = #next_motion.Data.PosLatchDistance.Edge
    DPLDti:
      REF = #next_motion.Data.PosLatchDistance.HwTrigIdx
    DPLDd:
      REF = #next_motion.Data.PosLatchDistance.Distance
    DPLli:
      REF = #next_motion.Data.PosLatch.LatchIdx
    DPLts:
      REF = #next_motion.Data.PosLatch.TriggSource
    DPLe:
      REF = #next_motion.Data.PosLatch.Edge
    DPLti:
      REF = #next_motion.Data.PosLatch.HwTrigIdx
    DPLtr:
      REF = #next_motion.Data.PosLatchGmc.Trigger
    DPLlp:
      REF = #next_motion.Data.PosLatchGmc.pLatchPos
    DPLcs:
      REF = #next_motion.Data.PosLatchGmc.CoordSystem
    DPLrp:
      REF = #next_motion.Data.PosLatchGmc.ResidualPath
    Drma:
      REF = #next_motion.Data.R_DependFeed.MaxRadius
    Drmi:
      REF = #next_motion.Data.R_DependFeed.MinRadius
    Drr:
      REF = #next_motion.Data.R_DependFeed.Rate
    Dsvp:
      SET = #next_motion.Data.Set_v_jump.programmed[0] = ArrayRep(:(:ncOFF:):);
        #next_motion.Data.Set_v_jump.programmed = ${EXPR};
    Dsvv:
      REF = #next_motion.Data.Set_v_jump.value
    Dsap:
      SET = #next_motion.Data.Set_a_jump.programmed[0] = ArrayRep(:(:ncOFF:):);
        #next_motion.Data.Set_a_jump.programmed = ${EXPR};
    Dsav:
      REF = #next_motion.Data.Set_a_jump.value
    Dsep:
      SET = #next_motion.Data.SetAxLimit.programmed[0] = ArrayRep(:(:ncOFF:):);
        #next_motion.Data.SetAxLimit.programmed = ${EXPR};
    Dser:
      REF = #next_motion.Data.SetAxLimit.RecordIdx
    Dcad:
      REF = #next_motion.Data.CamWrapping.Diameter
    Dcap:
      REF = #next_motion.Data.CamWrapping.ParameterP1
    Dsu:
      REF = #next_motion.Data.SetPathAccDec.UnitType
    Dsv108:
      SET = #next_motion.Data.SetPathAccDec.value = ${EXPR};
        if (#next_motion.Data.SetPathAccDec.UnitType == 1)
          %_CNC.lim_path_acc_p = ${EXPR} / 100.0 * %_CNC.lim_path_acc_p_ini;
        else
          %_CNC.lim_path_acc_p = ${EXPR};
        endif
    Dsv109:
      SET = #next_motion.Data.SetPathAccDec.value = ${EXPR};
        if (#next_motion.Data.SetPathAccDec.UnitType == 1)
          %_CNC.lim_path_acc_n = ${EXPR} / 100.0 * %_CNC.lim_path_acc_n_ini;
        else
          %_CNC.lim_path_acc_n = ${EXPR};
        endif
    Dsv110:
      SET = #next_motion.Data.SetPathAccDec.value = ${EXPR};
        if (#next_motion.Data.SetPathAccDec.UnitType == 1)
          %_CNC.lim_path_acc_p = ${EXPR} / 100.0 * %_CNC.lim_path_acc_p_ini;
          %_CNC.lim_path_acc_n = ${EXPR} / 100.0 * %_CNC.lim_path_acc_n_ini;
        else
          %_CNC.lim_path_acc_p = ${EXPR};
          %_CNC.lim_path_acc_n = ${EXPR};
        endif
    Daxlv:
      REF = #next_motion.Data.AxisLimit.Value
    Daxla:
      REF = #next_motion.Data.AxisLimit.Axis
    Daxlu:
      REF = #next_motion.Data.AxisLimit.UnitType
    Dsma:
      REF = #next_motion.Data.SetTransSpeed.MaxAngle
    Dsmi:
      REF = #next_motion.Data.SetTransSpeed.MinAngle
    Dsr:
      REF = #next_motion.Data.SetTransSpeed.RedFactor
    Dbrp:
      REF = #next_motion.Data.BezierSpline.RadiusProgrammed
    Dbr:
      REF = #next_motion.Data.BezierSpline.Radius
    Dbvp:
      REF = #next_motion.Data.BezierSpline.VeProgrammed
    Dbv:
      REF = #next_motion.Data.BezierSpline.Ve
    Dbl:
      REF = #next_motion.Data.BezierSpline.LinProgrammed
    Dbsf:
      REF = #next_motion.Data.BezierSpline.scalingFactor
    Dbsfd:
      REF = #next_motion.Data.BezierSpline.scalingFactor_def
    Dao:
      REF = #next_motion.Data.AutomTangentialAx.Offset
    Daa:
      REF = #next_motion.Data.AutomTangentialAx.AxIdx
    DAMa:
      REF = #next_motion.Data.AxisMapping.AxIdx
    DAMf:
      REF = #next_motion.Data.AxisMapping.factor
    DAMp:
      REF = #next_motion.Data.AxisMapping.ParameterP1
    DSPEid:
      REF = #next_motion.Data.SignalPathEnd.SignalId
    DSPEt:
      REF = #next_motion.Data.SignalPathEnd.Time
    DSPEst:
      REF = #next_motion.Data.SignalPathEnd.SignalType
    DSPEsi:
      REF = #next_motion.Data.SignalPathEnd.SignalIdx
    DSPEsd:
      REF = #next_motion.Data.SignalPathEnd.SourceData
    DSPEd:
      REF = #next_motion.Data.SignalPathEnd.DataLength
    DSPEp:
      SET = #next_motion.Data.SignalPathEnd.pDestination = \#sys_vars.EXF[0];
    DSPEDid:
      REF = #next_motion.Data.SignalPathEndDist.SignalId
    DSPEDd:
      REF = #next_motion.Data.SignalPathEndDist.Distance
    DSPEDst:
      REF = #next_motion.Data.SignalPathEndDist.SignalType
    DSPEDsi:
      REF = #next_motion.Data.SignalPathEndDist.SignalIdx
    DSPEDsd:
      REF = #next_motion.Data.SignalPathEndDist.SourceData
    DSPEDdl:
      REF = #next_motion.Data.SignalPathEndDist.DataLength
    DSPEDp:
      SET = #next_motion.Data.SignalPathEndDist.pDestination = \#sys_vars.EXF[0];
    DSPo:
      REF = #next_motion.Data.SignalPredict.Override
    DSPop:
      REF = #next_motion.Data.SignalPredict.OvrProgrammed
    DSPsi:
      REF = #next_motion.Data.SignalPredict.SignalIdx
    DSPsp:
      REF = #next_motion.Data.SignalPredict.StopProgrammed
    DWCx1:
      REF = #next_motion.Data.WS_Ctrl.x1
    DWCz1:
      REF = #next_motion.Data.WS_Ctrl.z1
    DWCy1:
      REF = #next_motion.Data.WS_Ctrl.y1
    DWCx2:
      REF = #next_motion.Data.WS_Ctrl.x2
    DWCz2:
      REF = #next_motion.Data.WS_Ctrl.y2
    DWCy2:
      REF = #next_motion.Data.WS_Ctrl.z2
    DWCi:
      REF = #next_motion.Data.WS_Ctrl.index
    DWCc:
      REF = #next_motion.Data.WS_Ctrl.coord
    DWCpl:
      REF = #next_motion.Data.WS_Ctrl.pplane
    DWCo:
      REF = #next_motion.Data.WS_Ctrl.orient
    DWCs:
      REF = #next_motion.Data.WS_Ctrl.shape
    DWCca:
      REF = #next_motion.Data.WS_Ctrl.clear_all
    DWCp1:
      REF = #next_motion.Data.WS_Ctrl.point1
    DWCp2:
      REF = #next_motion.Data.WS_Ctrl.point2
    DWCen:
      REF = #next_motion.Data.WS_Ctrl.enable
    DWCa:
      SET = #next_motion.Data.WS_Ctrl.arm_diameter[0] = ArrayRep(:(:ncOFF:):);
        #next_motion.Data.WS_Ctrl.arm_diameter = ${EXPR};
    DTDRt:
      REF = #next_motion.Data.ToolDataRecord.ToolIdx
    Sz:
      REF = #sys_vars.ZP
    DSSi:
      REF = #next_motion.Data.SpindleSpeed.Idx
    DSSs:
      REF = #next_motion.Data.SpindleSpeed.speed
    DCSSt:
      REF = #next_motion.Data.C2_SplineStart.BCType
    DCSSv:
      REF = #next_motion.Data.C2_SplineStart.BCValue
    DCSSp:
      SET = #next_motion.Data.C2_SplineStart.BCProgrammed[0] = ArrayRep(:(:ncOFF:):);
        #next_motion.Data.C2_SplineStart.BCProgrammed = ${EXPR};
    DCSSsp:
      REF = #next_motion.Data.C2_SplineStart.SegmentParameter
    DCSSst:
      REF = #next_motion.Data.C2_SplineStart.SegmentType
    DCSEt:
      REF = #next_motion.Data.C2_SplineEnd.BCType
    DCSEv:
      REF = #next_motion.Data.C2_SplineEnd.BCValue
    DCSEp:
      SET = #next_motion.Data.C2_SplineEnd.BCProgrammed[0] = ArrayRep(:(:ncOFF:):);
        #next_motion.Data.C2_SplineEnd.BCProgrammed = ${EXPR};
    DFd:
      REF = #next_motion.Data.Frame.Data
    DFcs:
      REF = #next_motion.Data.Frame.SetCS
    DSVs:
      REF = #next_motion.Data.SystemVariable.SysVarIdx
    DSVa:
      REF = #next_motion.Data.SystemVariable.AxIdx
    DSVd:
      REF = #next_motion.Data.SystemVariable.Data.R8_value
    DABNf:
      REF = #next_motion.Data.AutoBlockNumber.offset
    DABNo:
      REF = #next_motion.Data.AutoBlockNumber.factor
    DCSSPs:
      REF = #next_motion.Data.ConstantSurfaceSpeed.Speed
    DCSSPp:
      REF = #next_motion.Data.ConstantSurfaceSpeed.Programmed
    MXFPx:
      REF = #next_motion.Data.MXFrame.Pos.x
    MXFPy:
      REF = #next_motion.Data.MXFrame.Pos.y
    MXFPz:
      REF = #next_motion.Data.MXFrame.Pos.z
    MXFOt:
      REF = #next_motion.Data.MXFrame.Orient.Type
    MXFOa:
      REF = #next_motion.Data.MXFrame.Orient.Angle
    MXFEPx:
      REF = #next_motion.Data.MXFrameEx.Frame.Pos.x
    MXFEPy:
      REF = #next_motion.Data.MXFrameEx.Frame.Pos.y
    MXFEPz:
      REF = #next_motion.Data.MXFrameEx.Frame.Pos.z
    MXFEOt:
      REF = #next_motion.Data.MXFrameEx.Frame.Orient.Type
    MXFEOa:
      REF = #next_motion.Data.MXFrameEx.Frame.Orient.Angle
    MXFECs:
      REF = #next_motion.Data.MXFrameEx.SetCS
    MXFEAd:
      REF = #next_motion.Data.MXFrameEx.Additive
    MXTFPx:
      REF = #next_motion.Data.MXTool.Frame.Pos.x
    MXTFPy:
      REF = #next_motion.Data.MXTool.Frame.Pos.y
    MXTFPz:
      REF = #next_motion.Data.MXTool.Frame.Pos.z
    MXTFOt:
      REF = #next_motion.Data.MXTool.Frame.Orient.Type
    MXTFOa:
      REF = #next_motion.Data.MXTool.Frame.Orient.Angle
    MXTr:
      REF = #next_motion.Data.MXTool.Radius
    MXTi:
      REF = #next_motion.Data.MXTool.Index
    MXPPx:
      REF = #next_motion.Data.MXPoint.Pos.x
    MXPPy:
      REF = #next_motion.Data.MXPoint.Pos.y
    MXPPz:
      REF = #next_motion.Data.MXPoint.Pos.z
    MXPOt:
      REF = #next_motion.Data.MXPoint.Orient.Type
    MXPOa:
      REF = #next_motion.Data.MXPoint.Orient.Angle
    MXPCm:
      REF = #next_motion.Data.MXPoint.Cfg.Mode
    MXPr:
      REF = #next_motion.Data.MXPoint.RotAxis
    MXPa:
      REF = #next_motion.Data.MXPoint.AuxAxis
    MXPhTr:
      REF = #next_motion.Data.MXPathDesc.Trans.Radius
    MXPhTt:
      REF = #next_motion.Data.MXPathDesc.Trans.Type
    MXDa:
      REF = #next_motion.Data.MXDynamicDesc.Accel
    MXDd:
      REF = #next_motion.Data.MXDynamicDesc.Decel
    MXDOe:
      REF = #next_motion.Data.MXDynamicDesc.Optmot.Enable
    MXDOv:
      REF = #next_motion.Data.MXDynamicDesc.Optmot.VelPathDef
    MXDOr:
      REF = #next_motion.Data.MXDynamicDesc.Optmot.RobotPar
    MXDOl:
      REF = #next_motion.Data.MXDynamicDesc.Optmot.Limits
    MXVv:
      REF = #next_motion.Data.MXVelocity.v
    MXVm:
      REF = #next_motion.Data.MXVelocity.Mode
    MXAj:
      REF = #next_motion.Data.MXAxisTarget.JointAxis
    MXAa:
      REF = #next_motion.Data.MXAxisTarget.AuxAxis
    MXAb:
      REF = #next_motion.Data.MXAxisTarget.BaseAxis
    MXJ:
      REF = #next_motion.Data.MXJointAxis
    MXAto:
      REF = #next_motion.Data.MXAutoTang.Offset
    MXCDCas:
      REF = #next_motion.Data.MXCDC.ArcTransSpd
    MXCDCsm:
      REF = #next_motion.Data.MXCDC.SpdMode
    MXCDCcv:
      REF = #next_motion.Data.MXCDC.ContourViolation
    MXCDCtm:
      REF = #next_motion.Data.MXCDC.TransMode
    MXCDCem:
      REF = #next_motion.Data.MXCDC.EntryMode
    MXCDCal:
      REF = #next_motion.Data.MXCDC.AcrToLine
    THCp:
      REF = #next_motion.Data.ThreadCut.Position
    THCi:
      SET = #next_motion.Data.ThreadCut.Idx[0] = ArrayRep(:(:-1:):);
        #next_motion.Data.ThreadCut.Idx = ${EXPR};
    THCm:
      SET = #next_motion.Data.ThreadCut.Mode[0] = ArrayRep(:(:-1:):);
        #next_motion.Data.ThreadCut.Mode = ${EXPR};
    THCld:
      REF = #next_motion.Data.ThreadCut.LeadDirection
    THCl:
      REF = #next_motion.Data.ThreadCut.Lead
    THCo:
      REF = #next_motion.Data.ThreadCut.Offset
    ACVc:
      REF = #next_motion.Data.AxisCtrlVelocity.Command
    ACVi:
      REF = #next_motion.Data.AxisCtrlVelocity.Idx
    ACSs:
      REF = #next_motion.Data.AxisCtrlSpeed.Speed
    ACSi:
      REF = #next_motion.Data.AxisCtrlSpeed.Idx
    ACPp:
      REF = #next_motion.Data.AxisCtrlPosition.Position
    ACPd:
      REF = #next_motion.Data.AxisCtrlPosition.PositionDefined
    ACPi:
      REF = #next_motion.Data.AxisCtrlPosition.Idx
    ACPm:
      REF = #next_motion.Data.AxisCtrlPosition.Mode
    CHFm:
      REF = #next_motion.Data.Chamfer.Mode
    CHFv:
      REF = #next_motion.Data.Chamfer.Value
    PAFv:
      REF = #next_motion.Data.PathFeed.Value
    PAFi:
      REF = #next_motion.Data.PathFeed.Id
    GENd:
      REF = #next_motion.Data.GenericData.Data
    SGALda:
      REF = #next_motion.Data.SetGmcAxisLimit.DestinationAxis
    SGALdp:
      REF = #next_motion.Data.SetGmcAxisLimit.DestinationPath
    SGALsa:
      REF = #next_motion.Data.SetGmcAxisLimit.SourceAxis
    SGALsp:
      REF = #next_motion.Data.SetGmcAxisLimit.SourcePath
    SGALn:
      SET = BlockCpy(:\#next_motion.Data.SetGmcAxisLimit.SourceLimitSetName, ${EXPR}:);
    CMPmd:
      REF = #next_motion.Data.Compressor.MaxCartesianDeviation
    CMPmnd:
      REF = #next_motion.Data.Compressor.MaxNonCartesianDeviation
    CMPmt:
      REF = #next_motion.Data.Compressor.MaxCartesianTransitionAngle
    CMPml:
      REF = #next_motion.Data.Compressor.MaxCartesianLength
    CMPmnt:
      REF = #next_motion.Data.Compressor.MaxNonCartesianTransitionAngle
    PR8v:
      REF = #next_motion.Data.R8_param.Value
    PR8i:
      REF = #next_motion.Data.R8_param.Id
    STPi:
      REF = #next_motion.Data.ToolPar.Id
    STPR8:
      REF = #next_motion.Data.ToolPar.R8_value
    STPI4:
      REF = #next_motion.Data.ToolPar.I4_value
    GFof:
      REF = #next_motion.Data.GmcFrame.Offset
    GFmo:
      SET = #next_motion.Data.GmcFrame.Mode[0] = ArrayRep(:(:-1:):);
        #next_motion.Data.GmcFrame.Mode = ${EXPR};
    GFai:
      SET = #next_motion.Data.GmcFrame.AxIdx[0] = ArrayRep(:(:-1:):);
        #next_motion.Data.GmcFrame.AxIdx = ${EXPR};
    GFor:
      REF = #next_motion.Data.GmcFrame.Orientation
    GFori:
      SET = #next_motion.Data.GmcFrame.OrientationIdx[0] = ArrayRep(:(:-1:):);
        #next_motion.Data.GmcFrame.OrientationIdx = ${EXPR};
    GFort:
      REF = #next_motion.Data.GmcFrame.OrientationType
    GFsc:
      REF = #next_motion.Data.GmcFrame.SetCS
    GFtfc:
      REF = #next_motion.Data.GmcFrame.TCPFromCS
    GFttc:
      REF = #next_motion.Data.GmcFrame.TCPToCS
    GFcc:
      REF = #next_motion.Data.GmcFrame.ClearCS
    GFne:
      REF = #next_motion.Data.GmcFrame.Negative
    GFut:
      REF = #next_motion.Data.GmcFrame.UseTCP
  Constants:
    PathBusy = BUSY (type=STRING)
    PathStatus = STATUS (type=STRING)
    PathErrLevel = ERRLEV (type=STRING)
  BuiltInProcs:
    SendCommand = SendCommand(:$[1]:); (MinArgs=1, MaxArgs=1, Inline=Yes)
    DispatchAndWait = DispatchAndWait(:$[1]:); (MinArgs=1, MaxArgs=1, Inline=Yes)
    WaitForCommand = WaitForCommand(:$[1]:); (MinArgs=1, MaxArgs=1, Inline=Yes)
  Preprocess:
    MP_PJN (Search=MP22000 , Replace=PJN )
    MP_PJB (Search=MP22100 , Replace=PJB )
  GCodes:
    G_DELAY (GNum=0, Alias=@, AliasIsPattern=Yes, Inline=Yes)
      Arg (DataType=FLOAT, ref=tickdelay)
    G_PJN (GNum=22000, Alias=PJN, Group=220)
      Arg PathBusy (DataType=FLOAT, ref=busy_count)
      Arg PathStatus (DataType=FLOAT, ref=final_status)
      Arg PathErrLevel (DataType=FLOAT, ref=error_level)
    G_PJB (GNum=22100, Alias=PJB, Group=220)
      Arg PathBusy (DataType=FLOAT, ref=busy_count)
      Arg PathStatus (DataType=FLOAT, ref=final_status)
      Arg PathErrLevel (DataType=FLOAT, ref=error_level)
  MCodes:
    M_DEFAULT (IsDefault=Yes, MinValue=0, MaxValue=999999)
      ARG (ref=VALUE, DataType=FLOAT, RequireLiteral=Yes)
    M10003 = 10003 (Inline=Yes)
      ARG (ref=VALUE, DataType=FLOAT, RequireLiteral=Yes)
    M1000000 = 1000000 (Alias=;, AliasIsPattern=Yes, Inline=Yes, IgnoreIfGroups=220)
      ARG (ref=VALUE, DataType=FLOAT, RequireLiteral=Yes)
  ParserData (NestedComments=No, DefaultCaseSensitive=Yes, CommentsSpanLines=No, ReadWholeFileBeforeParsing=No, ExpectMainProgStmts=Yes, UseFubTemplates=No)
    TKG_END_OF_LINE = \n (IsPattern=No)
    TKG_OPEN_COMMENT = #
    TKG_NC_BLOCK_PREFIX = N:[\s\d] (IsPattern=Yes)
    TKG_OPEN_LISTBRACKET = (
    TKG_CLOSE_LISTBRACKET = )
    TKG_COMMA = ,
    TKG_NUMBER = \d+\.\d+|\d+\.|\.\d+ (IsPattern=Yes)
    TKG_INTEGER = \d+ (IsPattern=Yes)
    TKG_NUMBER_EXP = e:[\s\d\+\-\.] (IsPattern=Yes)
    TKG_ASSIGN_EQ = =
    TKG_ARITH_BINARY_MINUS = -
    TKG_M_CODE_PREFIX = MP:\d (IsPattern=Yes)
  StringChars (AsciiStringStart=")
    EscapeSeq (Search=$N, CaseSensitive=No, ReplaceValue=10)
    EscapeSeq (Search=$L, CaseSensitive=Yes, ReplaceValue=10)
    EscapeSeq (Search=$Q, CaseSensitive=No, ReplaceStr=")
    EscapeSeq (Search=$[\dA-F]+, IsPattern=Yes, CaseSensitive=No, ReplaceEncodingBase=16)
    EscapeSeq (Search=$$, ReplaceStr=$)
    EscapeSeq (Search=$, ReplaceStr=)
```

- Data object Logical/GmcIpConfig/gmcipesm (Cnc, version 5.02.1) (no source held here)

- Data object Logical/GmcIpConfig/gmcipmxd (Cnc, version 5.02.1) (no source held here)

### Data object Logical/GmcIpConfig/gmcipmx (Cnc, version 5.02.1)

#### gmcipmx.cnc
```
Root (LangModule=ailgcode, Version=1.0)
  AILHeader = sub OnProgStartPrivate
      %_Frm = %FRM_0;
      %_Base = %BASE_0;
      %_Tool = %TOOL_0;
      %_Vel = %VEL_0;
      %_Pth = %PTH_0;
      %_Dyn = %DYN_0;
      if (%_CNC.optmot_segmentation_on)
        %_Dyn.Optmot.Enable = 1 
      endif      
      BlockCpy(:\%_Ref, \%REF_0:);
    endsub
  BuiltInProcs:
    WAIT_PP_SYNC = #next_motion.Command = MPCMD_IP_SYNCH_PP;
      PushPacket(::);
      DispatchAndWait(:IPCMD_SYNC_PP_CONT:);
    ERROR_EX = ErrorEx(:"id":$[1],"fmt":$[2],"data":(:$[3],$[4],$[5],$[6],$[7],$[8],$[9],$[10],$[11],$[12],$[13],$[14]:):); (MinArgs=3, MaxArgs=14)
    SET_POINT:
      Arg (ref=POINT, DataType=ANY_DATA, MinCount=1, MaxCount=1)
    SET_TRIGGER_CONFIG:
      Arg (ref=TRIGGER, DataType=ANY_DATA, MinCount=1, MaxCount=1)
      Arg (ref=bHALT, DataType=ANY_DATA, MinCount=1, MaxCount=1)
      Arg (ref=ID, DataType=ANY_DATA, MinCount=1, MaxCount=1)
    SET_WANTED_JOINT:
      Arg (ref=Ref, DataType=ANY_DATA, MinCount=1, MaxCount=1)
    SET_CIRCLE:
      Arg (ref=END_POINT, DataType=ANY_DATA, MinCount=1, MaxCount=1)
      Arg (ref=CIRCLE_POINT, DataType=ANY_DATA, MinCount=1, MaxCount=1)
      Arg (ref=Angle, DataType=IEC_LREAL, MinCount=0, MaxCount=1)
    SET_AXIS_TARGET:
      Arg (ref=AXIS_TARGET, DataType=ANY_DATA, MinCount=1, MaxCount=1)
    SET_FRAME:
      Arg (ref=Frm, DataType=ANY_DATA, MinCount=0, MaxCount=1)
    SET_BASEFRAME:
      Arg (ref=Base, DataType=ANY_DATA, MinCount=0, MaxCount=1)
    SET_TOOL:
      Arg (ref=Tool, DataType=ANY_DATA, MinCount=0, MaxCount=1)
    SET_PATH_DESC:
      Arg (ref=Pth, DataType=ANY_DATA, MinCount=0, MaxCount=1)
    SET_DYNAMIC_DESC:
      Arg (ref=Dyn, DataType=ANY_DATA, MinCount=0, MaxCount=1)
    SET_VELOCITY:
      Arg (ref=Vel, DataType=ANY_DATA, MinCount=0, MaxCount=1)
    JointToPoint:
      Arg (ref=Joint, UserType=MXJointAxisType, MinCount=1, MaxCount=1)
      Arg (ref=Point, UserType=MXPointType, MinCount=1, MaxCount=1)
    PointToJoint:
      Arg (ref=Point, UserType=MXPointType, MinCount=1, MaxCount=1)
      Arg (ref=Joint, UserType=MXJointAxisType, MinCount=1, MaxCount=1)
    MoveL:
      Arg (ref=POINT, UserType=MXPointType, MinCount=1, MaxCount=1)
      Arg (ref=Frm, UserType=MXFrameType, MinCount=0, MaxCount=1)
      Arg (ref=Base, UserType=MXFrameType, MinCount=0, MaxCount=1)
      Arg (ref=Tool, UserType=MXToolType, MinCount=0, MaxCount=1)
      Arg (ref=Vel, UserType=MXVelocityType, MinCount=0, MaxCount=1)
      Arg (ref=Pth, UserType=MXPathDescType, MinCount=0, MaxCount=1)
      Arg (ref=Dyn, UserType=MXDynamicDescType, MinCount=0, MaxCount=1)
    MoveJ:
      Arg (ref=POINT, UserType=MXPointType, MinCount=1, MaxCount=1)
      Arg (ref=Frm, UserType=MXFrameType, MinCount=0, MaxCount=1)
      Arg (ref=Base, UserType=MXFrameType, MinCount=0, MaxCount=1)
      Arg (ref=Tool, UserType=MXToolType, MinCount=0, MaxCount=1)
      Arg (ref=Vel, UserType=MXVelocityType, MinCount=0, MaxCount=1)
      Arg (ref=Ref, UserType=MXJointAxisType, MinCount=0, MaxCount=1)
      Arg (ref=Pth, UserType=MXPathDescType, MinCount=0, MaxCount=1)
      Arg (ref=Dyn, UserType=MXDynamicDescType, MinCount=0, MaxCount=1)
    MoveC:
      Arg (ref=END_POINT, UserType=MXPointType, MinCount=1, MaxCount=1)
      Arg (ref=CIRCLE_POINT, UserType=MXPointType, MinCount=1, MaxCount=1)
      Arg (ref=Angle, DataType=IEC_LREAL, MinCount=0, MaxCount=1)
      Arg (ref=Frm, UserType=MXFrameType, MinCount=0, MaxCount=1)
      Arg (ref=Base, UserType=MXFrameType, MinCount=0, MaxCount=1)
      Arg (ref=Tool, UserType=MXToolType, MinCount=0, MaxCount=1)
      Arg (ref=Vel, UserType=MXVelocityType, MinCount=0, MaxCount=1)
      Arg (ref=Pth, UserType=MXPathDescType, MinCount=0, MaxCount=1)
      Arg (ref=Dyn, UserType=MXDynamicDescType, MinCount=0, MaxCount=1)
    MoveA:
      Arg (ref=AXIS_TARGET, UserType=MXAxisTargetType, MinCount=1, MaxCount=1)
      Arg (ref=Vel, UserType=MXVelocityType, MinCount=0, MaxCount=1)
      Arg (ref=Dyn, UserType=MXDynamicDescType, MinCount=0, MaxCount=1)
      Arg (ref=Pth, UserType=MXPathDescType, MinCount=0, MaxCount=1)
    MoveLSearch:
      Arg (ref=POINT, UserType=MXPointType, MinCount=1, MaxCount=1)
      Arg (ref=TRIGGER, UserType=MXTriggerConfigType, MinCount=1, MaxCount=1)
      Arg (ref=bHALT, DataType=IEC_BOOL, MinCount=1, MaxCount=1)
      Arg (ref=ID, DataType=IEC_UINT, MinCount=1, MaxCount=1)
      Arg (ref=Frm, UserType=MXFrameType, MinCount=0, MaxCount=1)
      Arg (ref=Base, UserType=MXFrameType, MinCount=0, MaxCount=1)
      Arg (ref=Tool, UserType=MXToolType, MinCount=0, MaxCount=1)
      Arg (ref=Vel, UserType=MXVelocityType, MinCount=0, MaxCount=1)
      Arg (ref=Pth, UserType=MXPathDescType, MinCount=0, MaxCount=1)
      Arg (ref=Dyn, UserType=MXDynamicDescType, MinCount=0, MaxCount=1)
    WaitTime:
      Arg (ref=set_time, DataType=IEC_LREAL, MinCount=1, MaxCount=1)
    WaitIp = #next_motion.Command = MPCMD_IP_SYNCH;
      if (#thread.restart.playback)
        #next_motion.Data.I4_value = ncSIMULATION;
      else
        #next_motion.Data.I4_value = ncSTANDARD;
      endif
      PushPacket(::);
      DispatchAndWait(:IPCMD_SYNC_PLC_CONT:);
    WaitEndMove = #next_motion.Command = MPCMD_IP_SYNCH_PATH;
      PushPacket(::);
      DispatchAndWait(:IPCMD_SYNC_PATH_CONT:);
    TmpTool = %__tmp_tool.Frame.Pos.x = %_CNC.tool_dx;
      %__tmp_tool.Frame.Pos.y = %_CNC.tool_dy;
      %__tmp_tool.Frame.Pos.z = %_CNC.tool_dz;
      %__tmp_tool.Frame.Orient.Type = %_CNC.tool_angles_type;
      %__tmp_tool.Frame.Orient.Angle[0] = %_CNC.tool_phi;
      %__tmp_tool.Frame.Orient.Angle[1] = %_CNC.tool_theta;
      %__tmp_tool.Frame.Orient.Angle[2] = %_CNC.tool_psi;
      %__tmp_tool.Frame.Orient.Angle[3] = 0;
      %__tmp_tool.Radius = #sys_vars.RAD;
    GetTool:
      Arg (ref=Tool, UserType=MXToolType, MinCount=1, MaxCount=1)
    TmpBaseFrame = %__tmp_frame.Pos.x = %_CNC.base_frame_dx;
      %__tmp_frame.Pos.y = %_CNC.base_frame_dy;
      %__tmp_frame.Pos.z = %_CNC.base_frame_dz;
      %__tmp_frame.Orient.Type = %_CNC.base_frame_angles_type;
      %__tmp_frame.Orient.Angle[0] = %_CNC.base_frame_phi;
      %__tmp_frame.Orient.Angle[1] = %_CNC.base_frame_theta;
      %__tmp_frame.Orient.Angle[2] = %_CNC.base_frame_psi;
      %__tmp_frame.Orient.Angle[3] = 0;
    GetBaseFrame:
      Arg (ref=Frame, UserType=MXFrameType, MinCount=1, MaxCount=1)
    GetJoint:
      Arg (ref=Joint, UserType=MXJointAxisType, MinCount=1, MaxCount=1)
    GetAxisTarget:
      Arg (ref=AxisTarget, UserType=MXAxisTargetType, MinCount=1, MaxCount=1)
    GetLatchPoint:
      Arg (ref=ID, DataType=IEC_UINT, MinCount=1, MaxCount=1)
      Arg (ref=Point, UserType=MXPointType, MinCount=1, MaxCount=1)
      Arg (ref=Event, DataType=IEC_BOOL, MinCount=1, MaxCount=1)
    GetPoint:
      Arg (ref=Point, UserType=MXPointType, MinCount=1, MaxCount=1)
    GetPointIntern = %__tmp_point = %POINT_0;
      
      local $i;
      $i=0;
      lbegin(1)
        %__tmp_axis_code[$i] = %_AX.axis_map[$i];
        %__tmp_axis_idx[$i] = %_AX.axis_map_idx[$i];
        $i = $i + 1;
      lend($i < GetIpInt(:300:))     
      %__mx_status =  MXCncAxesToPoint(:%_CNC.adr_trf_data_mx,  \%__tmp_set_pos, \%__tmp_point,   %_CNC.trf_type, %_CNC.angles_type, \%__tmp_axis_code, \%__tmp_axis_idx, GetIpInt(:300:) :);
      if (%__mx_status > 0)
        
        ErrorEx(:"id":10905,"fmt":"4d4d4d","data":(:GetCurLine(::),4,%__mx_status:):);
      endif
    CDCOn:
      Arg (ref=Direction, DataType=INT, MinCount=1, MaxCount=1)
      Arg (ref=CDC, UserType=MXCDCType, MinCount=0, MaxCount=1)
    CDCOff:
      Arg (ref=CDC, UserType=MXCDCType, MinCount=0, MaxCount=1)
    AutoTangOn:
      Arg (ref=Param, UserType=MXAutoTangType, MinCount=0, MaxCount=1)
    AutoTangOff = #next_motion.Command = MPCMD_MX_TANG_AX_OFF;
      PushPacket(::);
    SetM = local $i, $num_item;
      $i = 1;
      $num_item = ListLength(:${*}:);
      lbegin (1)
        #next_motion.Command = MPCMD_SET_M_FCT;
        #next_motion.Data.I4_value = ListItemValue(:${*}, $i:);  
        PushPacket(::);
        $i = $i + 1;
      lend($i <= $num_item)
      DispatchMPList(::); (MinArgs=1, MaxArgs=10)
  SysVars:
    TRF_DATA_MX $TRF_DATA_MX:
      GET = return %_CNC.adr_trf_data_mx; (ReturnType=IEC_UDINT)
```

- Data object Logical/GmcIpUserConfig/gmcipvar (Cnc, version 5.02.1) (no source held here)

- Data object Logical/GmcIpUserConfig/gmcipfun (Cnc, version 5.02.1) (no source held here)

- Data object Logical/GmcIpUserConfig/gmcipfub (Cnc, version 5.02.1) (no source held here)

- Data object Logical/GmcIpUserConfig/gmcipubr (Cnc, version 5.02.1) (no source held here)

- Data object Logical/GmcIpUserConfig/gmcipusm (Cnc, version 5.02.1) (no source held here)

- Data object Logical/GmcIpUserConfig/gmcipui (Cnc, version 5.02.1) (no source held here)

- Data object Logical/GmcIpUserConfig/gmcipus (Cnc, version 5.02.1) (no source held here)

- Data object Logical/GmcIpUserConfig/gmcipuc (Cnc, version 5.02.1) (no source held here)

Listed in the project but not available here: Logical/Global.typ, Logical/Libraries/Library1/Types.typ, Logical/Libraries/Library1/Constants.var, Logical/Types.typ
